Fanuc KAREL source: kt00893.KL

PROGRAM KT00893
%STACKSIZE=65535
%PRIORITY=65535
%NOLOCKGROUP
VAR
P1 : POSITION
P2 : POSITION
OUT : BOOLEAN
BEGIN
-- UNRESOLVED_PC line 8 opcodes [27 27 49 7E AD 27 9D 76 23] marker_code=0
END KT00893
